TYPE ST_AteqMapOutput :
STRUCT
	Write : ST_AteqMemoryToWrite;
END_STRUCT
END_TYPE

(* stored: Version 1.1.0.1
   DUT ST_AteqMapOutput: Id {176cd949-4a08-07c5-2535-3385e2e35db2} *)
